FUNCTION_BLOCK FB_Generator_Sine
VAR_INPUT
END_VAR
VAR_OUTPUT
END_VAR
VAR
END_VAR

END_FUNCTION_BLOCK

(* stored: Version 1.1.0.1, ProductVersion 3.1.4024.13
   POU FB_Generator_Sine: Id {e350ad4d-7b69-4ec8-912a-5345833cc920}, SpecialFunc None *)
